FUNCTION_BLOCK ABSTRACT FB_DS402Drive IMPLEMENTS I_DS402PiezoDrive
VAR_INPUT

END_VAR
VAR_OUTPUT

END_VAR
VAR
	{attribute 'no_copy'}
    stPiezoStage		:	REFERENCE TO ST_PiezoStage;
	eDriveState			:	E_DS402DriveState;
	fbLogError			:   FB_LogMotionError;
    eHomingState		: 	E_DS402Homing;
	// reuse to absolute/relative moves for DS402
    eAxisState			:  MC_AxisStates;
    // create a property for some of these
    bExecMove			: BOOL;
    bExecHome			: BOOL;
    bPosGoal			: BOOL;
    bNegGoal			: BOOL;
    bNewMoveReq			: BOOL;
    bHomingBusy			: BOOL;
    bHomingDone			: BOOL;
    bPrepareDisable		: BOOL;
    bMoveDone			: BOOL;
    bMoveBusy			: BOOL;
	bHalted				: BOOL;
	bAborted			: BOOL;
	bStopped			: BOOL;
	bServoOffTrans	: BOOL;
	bServoOnTrans : BOOL;
	bServoOffMode		:	BOOL ;
	bServoOnMode		: BOOL;
	bDiscreteInit		: BOOL;
	bDiscreteMotionAct  : BOOL;
	bServoOffparamsSet  : BOOL;
	bServoOffparamsSetDone : BOOL;
	bLimOverride				: BOOL;

    bError				: BOOL:=FALSE;
	bErrorStop			: BOOL;
    // use this for motion time axis states
    bExecute			: BOOL;
	// This prevent unexpected logical 1 on stMotionStage.bExecute 
    nErrorId			: UDINT:=0;
    sLocalErrorMessage	: STRING;
	nPiezoErrorCode		: UDINT;
	// Save abd restore encoder value
    bInit				: BOOL;
    bLoad				: BOOL;
    bEncError			: BOOL;
	bSaveDone			: BOOL;
	bAbortDone			: BOOL;
    // axis status -- emulating some NC axis
    bClosedLoopMode		:	BOOL;
    bPositiveDirection	:  	BOOL;
    bNegativeDirection 	:  	BOOL;
    bInTargetPosition 	:  	BOOL;
	bReadErrDone			: 	BOOL;
	bLogReady			: 	BOOL;
	bFault				: 	BOOL;
    bDiscreteMotion 	:  	BOOL;
    bContinuousMotion 	:  	BOOL;

    bSlowParamReadTimer	: 	BOOL := TRUE;
	
    // Drive calibrated motion params
    nCalibratedVelocity			: DINT;
    nCalibratedAcceleration		: DINT;
    nCalibratedTargetPosition 	: DINT;
    nCalibratedMaxVelocity 		: DINT;
    nCalibratedMaxAcceleration	: DINT;
    nCalibratedHomeVelocity 	: DINT;
    nCalibratedHomeAcceleration	: DINT;

	// Open Loop Motion paramters
    nCalibratedSteps			: DINT;
    nCalibratedStepAmp			: UINT;
    nCalibratedStepFreq 		: UINT;

    // Calibrated motion params : nanometer operation by default.
    fCalibratedStandStillPos	: REAL;
    fOverride					: REAL;
	fDefaultScalingFactor 		: REAL:=0.000001;
    fCalibratedActPos			: REAL;
	rtHaltedDone	: R_TRIG;
	rtTargetReached	: R_TRIG;
	ftAbortDone: F_TRIG;
	rtFault			: R_TRIG;
    rtHomed			: R_TRIG;
    rtMoveCmdShortcut	: R_TRIG;
    rtHomeCmdShortcut	: R_TRIG;
    rtEnableMode		: R_TRIG;
    rtUserExec			: R_TRIG;
	rtErrorStop			: R_TRIG;
    rtTarget		: R_TRIG;
	rtServoOnMode	: R_TRIG;
    rtEnableDrive	: R_TRIG;
	rtServoOnTrans	: R_TRIG;
	rtNotClState 	: R_TRIG;
	rtNotOlState 	: R_TRIG;
	rtNewMoveReq	: R_TRIG;

	ftServoOffTrans	: F_TRIG;
	rtServoOffMode	: R_TRIG;
	ftAmsNetId 		: F_TRIG;
    ftExec			: F_TRIG;
	ftErrorSdoRead	: F_TRIG;
    ftEnableDrive	: F_TRIG;
	ftForwardEnabled	: F_TRIG;
	ftBackwardEnabled	: F_TRIG;
	ftServo				: F_TRIG;
	
    ftSdoStep		: 	F_TRIG;
    ftSdoStepFreq	: 	F_TRIG;
    ftSdoStepAmp	: 	F_TRIG;
	
    tonSyncHoming 		: TON;
	tonHoldTime			: TON;
	tonServoOffSync		: TON;
    tonSlowParamReadTimer: TON;
	// fast changing paramter timer -- wwe could have used PDO for this params
	// but the Piezo ESC have fixed PDO list.
	tonFastParamReadTimer: TON;
	//bInitiated	: BOOL;
    // Diagnotics data from the drive, mainly Error codes
	tRefreshDelay   : TIME := T#1S;
	tSavedholtime	: TIME;
	// Open Loop Operations
    fbSdoStep		: 	FB_EcCoESdoWrite;
    fbSdoStepFreq	: 	FB_EcCoESdoWrite;
    fbSdoStepAmp	: 	FB_EcCoESdoWrite;
	
    fbErrorSdoRead			: FB_EcCoESdoRead;
    fbFollowWinSdoRead		: FB_EcCoESdoRead;
    fbSoftLimMaxSdoRead		: FB_EcCoESdoRead;
    fbSoftLimMinSdoRead 	: FB_EcCoESdoRead;
    fbMotorloadSdoRead		: FB_EcCoESdoRead;
    fbGetAmsNetId			: FB_GetLocalAmsNetId;

    sAmsNetId 				: T_AmsNetId;
    nSubIndex  				: BYTE := 0;

  	nChanFErrWinIdx		: WORD;
  	nChanSoftwareLimIdx	: WORD;
  	nChanMotorLoadIdx	: WORD;
	nChanErrorCodeIdx	: WORD;
    nChanOlStepIdx		: WORD;
    nChanOlStepFreqIdx	: WORD;
    nChanOlStepAmpIdx	: WORD;

    nChanPrevStep			: DINT;
    nChanPrevStepFreq		: UINT;
    nChanPrevStepAmp		: UINT;

	
END_VAR


VAR CONSTANT
    nScaleOffsetBase	: WORD := 16#2007;
    nScaleInvBase		: WORD := 16#2008;
	nMotorLoadbase		: WORD := 16#200d;
    nSoftLimBase		: WORD := 16#200e;
	nHomeOffsetBase		: WORD := 16#607C;
	nHomingSpeedBase	: WORD := 16#6099;
	nhomingAccBase		: WORD := 16#609a;
	nErrorCodeBase		: WORD := 16#603f;
	nFErrWinBase		: WORD := 16#6065;
	nOlStepBase		: WORD := 16#2022;
	nOlStepAmpBase		: WORD := 16#2023;
	nOlStepFreqBase	: WORD := 16#2024;
	// this true for SmartAct MCS2 and E-727.
	nChanOfsBase	: WORD := 16#800;
	// DS 402 Motor encoder defective code : this is needed for save and restore.
	nEncErrorCode	: WORD := 16#7300;

END_VAR


VAR PERSISTENT
    bSaved: BOOL;
    fPosition: LREAL;
END_VAR

{attribute 'monitoring':= 'variable'}
PROPERTY AbortDone : BOOL
GET
AbortDone:=bAbortDone;
END_GET
SET
bAbortDone := AbortDone;
END_SET
END_PROPERTY

{attribute 'monitoring':= 'variable'}
PROPERTY Aborted : BOOL
GET
Aborted := bAborted;
END_GET
SET
bAborted := Aborted;
END_SET
END_PROPERTY

METHOD AmsNetIdToString
VAR_INPUT

END_VAR

VAR
	nCounter: UINT;
	sAmsNetTmp: STRING(255);
END_VAR
IF sAmsNetId = '' THEN
	FOR nCounter := 0 TO (SIZEOF(stPiezoStage.arNetId)-1) BY 1 DO
		IF nCounter <= ((SIZEOF(stPiezoStage.arNetId)-1) -1) THEN
			sAmsNetTmp := CONCAT(BYTE_TO_STRING(stPiezoStage.arNetId[nCounter]),'.');
		ELSE
			sAmsNetTmp := BYTE_TO_STRING(stPiezoStage.arNetId[nCounter]);
		END_IF
		sAmsNetId := CONCAT(sAmsNetId, sAmsNetTmp);
	END_FOR	
END_IF
END_METHOD

METHOD PUBLIC ABSTRACT Brake
END_METHOD

PROPERTY CalibratedAcceleration : DINT
GET
CalibratedAcceleration:=nCalibratedAcceleration;
END_GET
END_PROPERTY

PROPERTY CalibratedActPos : REAL
GET
CalibratedActPos:=fCalibratedActPos;
END_GET
END_PROPERTY

PROPERTY CalibratedHomeAcceleration : DINT
GET
CalibratedHomeAcceleration:= nCalibratedHomeVelocity;
END_GET
END_PROPERTY

PROPERTY CalibratedHomeVelocity : DINT
GET
CalibratedHomeVelocity:=nCalibratedHomeVelocity;
END_GET
END_PROPERTY

PROPERTY CalibratedMaxAcceleration : DINT
GET
CalibratedMaxAcceleration:= nCalibratedMaxAcceleration;
END_GET
END_PROPERTY

PROPERTY CalibratedMaxVelocity : DINT
GET
CalibratedMaxVelocity:= nCalibratedMaxVelocity;
END_GET
END_PROPERTY

METHOD CalibratedServoOnParams
VAR_INPUT
END_VAR
VAR

END_VAR
// All drive paramters must be express in mm, mm/s, mm/s2
nCalibratedMaxVelocity:=REAL_TO_DINT((stPiezoStage.fMaxVelocity / MAX(stPiezoStage.fscalingFactor, fDefaultScalingFactor)));
nCalibratedMaxAcceleration:=LREAL_TO_DINT(stPiezoStage.fMaxAcceleration /  MAX(stPiezoStage.fscalingFactor, fDefaultScalingFactor));
// Homing params
nCalibratedHomeVelocity:=LIMIT(0, LREAL_TO_DINT (stPiezoStage.fVelocity / MAX(stPiezoStage.fscalingFactor, fDefaultScalingFactor)), nCalibratedMaxVelocity);
nCalibratedHomeAcceleration:=LIMIT(0, LREAL_TO_DINT (stPiezoStage.fAcceleration / MAX(stPiezoStage.fscalingFactor, fDefaultScalingFactor)), nCalibratedMaxAcceleration) ;
// Target Position
nCalibratedTargetPosition:=LREAL_TO_DINT (stPiezoStage.fPosition / MAX(stPiezoStage.fscalingFactor, fDefaultScalingFactor));
// set soft limit on drive params to avoid bumping hard on the end stops
nCalibratedVelocity:=LIMIT(0, LREAL_TO_DINT (stPiezoStage.fVelocity / MAX(stPiezoStage.fscalingFactor, fDefaultScalingFactor)), nCalibratedMaxVelocity);
nCalibratedAcceleration:=LIMIT(0, LREAL_TO_DINT (stPiezoStage.fAcceleration / MAX(stPiezoStage.fscalingFactor, fDefaultScalingFactor)), nCalibratedMaxAcceleration) ;
END_METHOD

PROPERTY CalibratedTargetPosition : DINT
GET
CalibratedTargetPosition:= nCalibratedTargetPosition;
END_GET
END_PROPERTY

PROPERTY CalibratedVelocity : DINT
GET
CalibratedVelocity:=nCalibratedVelocity;
END_GET
END_PROPERTY

METHOD CalibrateServoOffParams
VAR_INPUT
END_VAR
// Open Loop Step Mode parameters
nCalibratedSteps:=LIMIT(-100000, stPiezoStage.nChanStep, 100000);
nCalibratedStepAmp:=REAL_TO_UINT(LIMIT(1, stPiezoStage.nChanStepAmp, 100) * 655.35);
nCalibratedStepFreq:=REAL_TO_UINT(LIMIT(1.0, stPiezoStage.nChanStepFreq, 1000.0));
END_METHOD

METHOD EncSaveRestore
VAR_INPUT
	bEnable	: BOOL;
END_VAR
IF bEnable THEN
    // Trigger a load if anything was saved at all
    IF NOT bInit THEN
        bInit := TRUE;
        bLoad S= bSaved;
    END_IF

    // Set our position if bLoad is true
	IF bLoad THEN
		stPiezoStage.fPosition:=fPosition;
		bSaveDone := TRUE;
	END_IF

    // Only load once, at startup
    bLoad R= bSaveDone;

    // Check ST_PiezoStage for an encoder error
    bEncError := stPiezoStage.bError AND (stPiezoStage.nErrorId = nEncErrorCode);

    // Do not save if we're currently loading or if there is an encoder error
    IF NOT bLoad AND NOT bEncError THEN
        fPosition := stPiezoStage.stAxisStatus.fActPosition;
        // This persistent variable lets us check if anything was saved
        // It will be TRUE at startup if we have saved values
        bSaved := TRUE;
    END_IF
END_IF
END_METHOD

METHOD EncValue
VAR_INPUT
  //  bEnable: BOOL;
END_VAR
(* SmartACT: The encoder count from the Piezo drive is not a raw count from the embeded actuator device
   we get a calibrated nm value. thus the use of abs() since this value is signed. 
   PI: to be discovered *)
IF stPiezoStage.nRawEncoderDINT <> 0 THEN
    stPiezoStage.nEncoderCount:=DINT_TO_UDINT(ABS(stPiezoStage.nRawEncoderDINT));
ELSE
    stPiezoStage.nEncoderCount:=0;
END_IF

// calibrated encoder readback
fCalibratedActPos:=DINT_TO_REAL(stPiezoStage.nRawEncoderDINT) *  MAX(stPiezoStage.fscalingFactor, fDefaultScalingFactor);
stPiezoStage.fPosDiff:=ABS(stPiezoStage.fPosition) - ABS(fCalibratedActPos);
END_METHOD

{attribute 'monitoring':= 'variable'}
PROPERTY Error : BOOL
GET
Error:=bError;
END_GET
SET
bError:=Error;
END_SET
END_PROPERTY

{attribute 'monitoring':= 'variable'}
PROPERTY ErrorCode : UDINT
GET
ErrorCode:=nErrorID;
END_GET
SET
nErrorID:=ErrorCode;
END_SET
END_PROPERTY

PROPERTY ErrorMessage : STRING
GET
ErrorMessage:=sLocalErrorMessage;
END_GET
SET
sLocalErrorMessage:=ErrorMessage;
END_SET
END_PROPERTY

//FB_Init is always available implicitly and it is used primarily for initialization.
//The return value is not evaluated. For a specific influence, you can also declare the
//methods explicitly and provide additional code there with the standard initialization
//code. You can evaluate the return value.
METHOD FB_Init: BOOL
VAR_INPUT
    bInitRetains: BOOL; // TRUE: the retain variables are initialized (reset warm / reset cold)
    bInCopyCode: BOOL;  // TRUE: the instance will be copied to the copy code afterward (online change)   
    stPzStage		:	REFERENCE TO ST_PiezoStage;
END_VAR
stPiezoStage REF= stPzStage;
END_METHOD

METHOD GetAmsNetId : BOOL
VAR_INPUT
	isNotSet : BOOL;
END_VAR

VAR
	
END_VAR
ftAmsNetId(CLK:=fbGetAmsNetId.bBusy);

fbGetAmsNetId(bExecute := isNotSet, tTimeOut := T#2S);

IF ftAmsNetId.Q  THEN
	IF NOT fbGetAmsNetId.bError THEN
		sAmsNetId := fbGetAmsNetId.AddrString;
	ELSE
		Error := fbGetAmsNetId.bError;
		ErrorCode := fbGetAmsNetId.nErrId;
	END_IF
	fbGetAmsNetId.bExecute := FALSE;
END_IF
END_METHOD

METHOD Halt : BOOL


Stopped S= NOT Error AND MoveBusy AND (stPiezoStage.bHalt OR NOT stPiezoStage.bExecute);

stPiezoStage.nPiezoDriveControl.8 := Stopped;
END_METHOD

{attribute 'monitoring':= 'variable'}
PROPERTY Halted : BOOL
GET
Halted := bHalted;
END_GET
SET
bHalted := Halted;
END_SET
END_PROPERTY

METHOD ABSTRACT HandleMoveRequest
VAR_INPUT
END_VAR
END_METHOD

METHOD PUBLIC Home : BOOL
tonSyncHoming(PT:=T#1000MS);
(* IMPORTANT: Homing options and parameters must be configured either via the COE online tab or via the service tool *)
CASE eHomingState OF
    E_DS402Homing.INIT_HOMING :;
        stPiezoStage.nModeOfOperation:=E_DS402OpMode.HOMING;
        IF stPiezoStage.nModeOfOperationDisplay = E_DS402OpMode.HOMING THEN
			HomeDone := FALSE;
			tonSyncHoming.IN := TRUE;
            stPiezoStage.nPiezoDriveControl.4:=TRUE;
			IF tonSyncHoming.Q THEN
				eHomingState:=E_DS402Homing.HOMING_IN_PROGRESS;
			END_IF
        END_IF

    E_DS402Homing.HOMING_IN_PROGRESS:
        IF NOT stPiezoStage.stPiezoDriveStatus.TargetReached
           AND NOT stPiezoStage.stPiezoDriveStatus.Bit13_OpModeSpecific THEN
                HomingBusy:=TRUE;
                HomeDone:=FALSE;
        END_IF
		
        // Interrupted
        IF stPiezoStage.stPiezoDriveStatus.TargetReached 
			AND NOT stPiezoStage.stPiezoDriveStatus.Bit12_OpModeSpecific THEN
            eHomingState:=E_DS402Homing.HOMING_INTERRUPTED;
        END_IF

        // Reached
        IF stPiezoStage.stPiezoDriveStatus.TargetReached
            AND stPiezoStage.stPiezoDriveStatus.Bit12_OpModeSpecific
            AND NOT stPiezoStage.stPiezoDriveStatus.Bit13_OpModeSpecific THEN
            eHomingState:=E_DS402Homing.HOMING_ATTAINED;
        END_IF

    E_DS402Homing.HOMING_ATTAINED:;
        HomingBusy:=FALSE;
        HomeDone:=TRUE;
        Error:=FALSE;
		tonSyncHoming.IN := FALSE;
		stPiezoStage.fPosition := 0.0;
		//prepare next move
		stPiezoStage.nPiezoDriveControl.4:=FALSE;
		stPiezoStage.nModeOfOperation:=E_DS402OpMode.PROFILE_POSITION;
		
    E_DS402Homing.HOMING_INTERRUPTED :;
        HomingBusy:=FALSE;
        HomeDone:=FALSE;
        ErrorMessage:='Warning: Halt interrupted homing sequence';
        Error:=FALSE;
        ErrorCode:=99; 

END_CASE
END_METHOD

{attribute 'monitoring':= 'variable'}
PROPERTY HomeDone : BOOL
GET
HomeDone:=bHomingDone;
END_GET
SET
bHomingDone:=HomeDone;
END_SET
END_PROPERTY

{attribute 'monitoring':= 'variable'}
PROPERTY HomingBusy : BOOL
GET
HomingBusy:=bHomingBusy;
END_GET
SET
bHomingBusy:=HomingBusy;
END_SET
END_PROPERTY

{attribute 'monitoring':= 'variable'}
PROPERTY PROTECTED InTargetPosition : BOOL
GET
 InTargetPosition := bInTargetPosition;
END_GET
SET
 bInTargetPosition := InTargetPosition;
END_SET
END_PROPERTY

METHOD PUBLIC Interlock

VAR
END_VAR
// Check for the plc shortcut commands
// Used for testing or to circumvent motor record issues
rtMoveCmdShortcut(CLK:=stPiezoStage.bMoveCmd);
rtHomeCmdShortcut(CLK:=stPiezoStage.bHomeCmd);

// Execute on rising edge
IF rtMoveCmdShortcut.Q AND NOT stPiezoStage.bExecute THEN
    stPiezoStage.bExecute:=TRUE;
    stPiezoStage.nCommand:=E_EpicsMotorCmd.MOVE_ABSOLUTE;
    // attempting to move an axis without homing first?
    IF stPiezoStage.nHomingMode <> E_EpicsHomeCmd.NONE AND NOT stPiezoStage.bHomed THEN
        // one can just set bHome here even though no homing was done?
        stPiezoStage.sErrorMessage:='Axis homing mode set, but homing routine pending';
    END_IF

ELSIF rtHomeCmdShortcut.Q AND NOT stPiezoStage.bExecute THEN
    stPiezoStage.bExecute:= NOT ( stPiezoStage.nCmdData = E_EpicsHomeCmd.ABSOLUTE_SET ) OR NOT ( stPiezoStage.nCmdData = E_EpicsHomeCmd.NONE);

    stPiezoStage.nCommand:=E_EpicsMotorCmd.HOME;
	// Automatically fill the correct nCmdData for homing
	stPiezoStage.nCmdData:=stPiezoStage.nHomingMode;
END_IF

// Handle main execs .  Rising on bMoved should be the ntry point
// bu this is not the case in production its a rising on bExecute.
rtUserExec(CLK:=stPiezoStage.bExecute);
// if a Move/Home Goal is comfirmed and there is no persistant 
// error conditions, then we have a valid move request.
bNewMoveReq S= NOT stPiezoStage.stAxisStatus.bBusy AND rtUserExec.Q AND NOT stPiezoStage.bError;
// this Move request is valid till an error occurs or the currently move is done
bNewMoveReq R= NOT stPiezoStage.bExecute OR stPiezoStage.bError;
bPrepareDisable R= bNewMoveReq;
// define this R_TRIG to comfirm a new move request.
rtNewMoveReq(CLK:=bNewMoveReq);
// Moves are automatically allowed if no safety hooks. Otherwise, some other code will set this.
stPiezoStage.bSafetyReady S= stPiezoStage.bPowerSelf;

// Transition to DURING_MOTION drive mode
rtEnableMode(CLK:=(stPiezoStage.nEnableMode = E_StageEnableMode.DURING_MOTION));
// Handle auto-enable timing
CASE stPiezoStage.nEnableMode OF
    E_StageEnableMode.ALWAYS:
        stPiezoStage.bEnable:=TRUE;
    E_StageEnableMode.DURING_MOTION:
		IF rtEnableMode.Q THEN
			stPiezoStage.bEnable := FALSE;
		END_IF
		// Power only enabled with a new move request
		IF rtNewMoveReq.Q THEN
			stPiezoStage.bEnable S= stPiezoStage.bSafetyReady;
		END_IF
END_CASE

bPosGoal  S= rtNewMoveReq.Q AND (stPiezoStage.stAxisStatus.fActPosition < stPiezoStage.fPosition) ;
bNegGoal  S= rtNewMoveReq.Q AND (stPiezoStage.stAxisStatus.fActPosition > stPiezoStage.fPosition) ;

bPosGoal  R= HomingBusy OR bNegGoal;
bNegGoal  R= HomingBusy OR bPosGoal;
// use falling trigger to avoid spaming  sErrorMessage
ftForwardEnabled(CLK:=stPiezoStage.bAllForwardEnable);
ftBackwardEnabled(CLK:=stPiezoStage.bAllBackwardEnable);

IF  NOT HomingBusy AND ftForwardEnabled.Q THEN
	// Not an error, just a warning
	stPiezoStage.sErrorMessage:='Cannot move past positive limit.';
	bLimOverride := TRUE;
	stPiezoStage.bExecute:=FALSE;
END_IF
	
IF NOT HomingBusy AND ftBackwardEnabled.Q THEN
	// Not an error, just a warning
	stPiezoStage.sErrorMessage:='Cannot move past Negative limit.';
	bLimOverride := TRUE;
	stPiezoStage.bExecute:=FALSE;
END_IF

IF NOT stPiezoStage.bError AND stPiezoStage.bExecute AND NOT stPiezoStage.bUserEnable THEN
    stPiezoStage.bError := TRUE;
    stPiezoStage.nErrorId := 1;
    stPiezoStage.sCustomErrorMessage := 'Move requested, but user enable is disabled!';
END_IF

// Update all enable booleans
SetEnables();

CASE McAxisState OF
    // We are not enabled if there is an issue
    MC_AXISSTATE_UNDEFINED, MC_AXISSTATE_DISABLED, MC_AXISSTATE_ERRORSTOP:
        stPiezoStage.bEnableDone:=FALSE;
    ELSE
        stPiezoStage.bEnableDone:=TRUE;
END_CASE

bExecute:= NOT stPiezoStage.bError AND stPiezoStage.bExecute AND stPiezoStage.bAllEnable AND stPiezoStage.bEnableDone AND stPiezoStage.bSafetyReady;
// 
bExecHome:=bExecute AND stPiezoStage.nCommand = 10;
bExecMove:=bExecute AND NOT bExecHome;

(*  *)
ftExec(CLK:=stPiezoStage.bExecute);
END_METHOD

METHOD PUBLIC Logger
END_METHOD

{attribute 'monitoring':= 'variable'}
PROPERTY McAxisState : MC_AxisStates
GET
McAxisState := eAxisState;
END_GET
SET
eAxisState := McAxisState;
END_SET
END_PROPERTY

METHOD PUBLIC  MotionParams
VAR_INPUT
    tRefreshDelay: TIME;
END_VAR
// get periodique update on Motion params
ReadDriveParams();
// 
// Copy axis parameters that we want to expose to the EPICS layer.
stPiezoStage.stAxisParametersExposed.bCtrlEnablePosDiffControl     := stPiezoStage.stAxisParameters.bCtrlEnablePosDiffControl;
stPiezoStage.stAxisParametersExposed.bEncEnableSoftEndMaxControl   := stPiezoStage.stAxisParameters.bEncEnableSoftEndMaxControl ;
stPiezoStage.stAxisParametersExposed.bEncEnableSoftEndMinControl   := stPiezoStage.stAxisParameters.bEncEnableSoftEndMinControl;
stPiezoStage.stAxisParametersExposed.fAccelerationMax              := stPiezoStage.stAxisParameters.fAccelerationMax;
stPiezoStage.stAxisParametersExposed.fCtrlPosDiffMax               := stPiezoStage.stAxisParameters.fCtrlPosDiffMax;
stPiezoStage.stAxisParametersExposed.fCtrlPosDiffMaxTime           := stPiezoStage.stAxisParameters.fCtrlPosDiffMaxTime;
stPiezoStage.stAxisParametersExposed.fDecelerationMax              := stPiezoStage.stAxisParameters.fDecelerationMax;
stPiezoStage.stAxisParametersExposed.fEncSoftEndMax                := stPiezoStage.stAxisParameters.fEncSoftEndMax;
stPiezoStage.stAxisParametersExposed.fEncSoftEndMin                := stPiezoStage.stAxisParameters.fEncSoftEndMin;
stPiezoStage.stAxisParametersExposed.fVeloMaximum                  := stPiezoStage.stAxisParameters.fVeloMaximum;
stPiezoStage.stAxisParametersExposed.fEncOffset               	  := stPiezoStage.stAxisParameters.fEncOffset;
stPiezoStage.stAxisParametersExposed.fEncScaleFactorInternal       := stPiezoStage.stAxisParameters.fEncScaleFactorInternal;
END_METHOD

METHOD PUBLIC ABSTRACT MoveAbsolute
END_METHOD

{attribute 'monitoring':= 'variable'}
PROPERTY MoveBusy : BOOL
GET
MoveBusy:=bMoveBusy;
END_GET
SET
bMoveBusy:=MoveBusy;
END_SET
END_PROPERTY

{attribute 'monitoring':= 'variable'}
PROPERTY MoveDone : BOOL
GET
MoveDone:=bMoveDone;
END_GET
SET
bMoveDone:=MoveDone;
END_SET
END_PROPERTY

METHOD PUBLIC ABSTRACT MoveRelative
VAR_INPUT
END_VAR
END_METHOD

METHOD PUBLIC ABSTRACT MoveVelocity
END_METHOD

{attribute 'monitoring':= 'variable'}
PROPERTY PiezoErrorCode : UDINT
GET
PiezoErrorCode := nPiezoErrorCode;
END_GET
SET
nPiezoErrorCode := PiezoErrorCode;
END_SET
END_PROPERTY

METHOD PostInterlocks
VAR_INPUT
END_VAR
// user override aka stop from EPICS ?
// Check done moving via user stop, fbDriveVirtual and Target Position Monitoring, or from homing.
// set/reset stPiezoStage.bDone after move absolute/Relative

// need to catch this as soon as it happen and must be seen by every call after intelock()
// within the sma ecycle
ftAbortDone(CLK:=AbortDone);
//rtErrorStop(CLK:=bErrorStop);

rtTarget(CLK:=(InTargetPosition AND MoveDone AND bExecMove));
rtHomed(CLK:=HomeDone AND bExecHome);
IF (*rtErrorStop.Q OR*) ftAbortDone.Q OR  rtTarget.Q OR rtHomed.Q THEN
    IF NOT stPiezoStage.bDone THEN
		MoveBusy:=FALSE;
		stPiezoStage.bDone := MoveDone OR HomeDone;
		stPiezoStage.bHomed := HomeDone;
		AbortDone := FALSE;
		bErrorStop:=FALSE;
        IF NOT Error THEN
            bExecute:=FALSE;
            stPiezoStage.bExecute:=FALSE;
        END_IF
    END_IF
END_IF

IF bExecute AND NOT Error THEN
    // Reset local warnings if things are going well
    stPiezoStage.sErrorMessage:='';
END_IF

// Handle auto-disable timing
bPrepareDisable S= stPiezoStage.nEnableMode = E_StageEnableMode.DURING_MOTION AND ftExec.Q;
// Delay the disable until we reach standstill, else brake issues or other race conditions
IF bPrepareDisable AND eAxisState = MC_AXISSTATE_STANDSTILL THEN
    bPrepareDisable:=FALSE;
    stPiezoStage.bEnable:=FALSE;
END_IF

//---------- brakes code here ---------------

// Always reset, even if not rising edge, so command can be issued again
// but do so only after the move was done or was cancel due to error or an interlock condition
IF ftExec.Q AND (stPiezoStage.bMoveCmd OR stPiezoStage.bHomeCmd) THEN
    stPiezoStage.bMoveCmd:=FALSE;
    stPiezoStage.bHomeCmd:=FALSE;

END_IF

// Force everything off in case of error
IF stPiezoStage.bError THEN
    stPiezoStage.bBusy := FALSE;
    stPiezoStage.bDone := FALSE;
    stPiezoStage.bEnable := FALSE;
END_IF

stPiezoStage.bBusy:=HomingBusy OR MoveBusy;

// Log errors
// Set the error message if we have one

// Hook if other code wants to inject a non-NC error
IF stPiezoStage.sCustomErrorMessage <> '' THEN
	bLogReady := FALSE;
	stPiezoStage.sErrorMessage := stPiezoStage.sCustomErrorMessage;

ELSE
	stPiezoStage.sErrorMessage := F_MotionErrorCodeLookup(nErrorId := stPiezoStage.nErrorId);
END_IF

fbLogError( stMotionStage:=stPiezoStage, bEnable:=bLogReady);
END_METHOD

METHOD Power : BOOL
// No transition while the drive is in motion
// transition from close to open loop. while moving

rtEnableDrive(CLK:=stPiezoStage.bAllEnable);
ftEnableDrive(CLK:=stPiezoStage.bAllEnable);

ftServoOffTrans(CLK:=(NOT bFault AND stPiezoStage.bServo));
rtServoOnTrans(CLK:=(NOT bFault AND stPiezoStage.bServo));

//rtServoOffMode(CLK:=bServoOffMode);
//rtServoOnMode(CLK:=stPiezoStage.bAllEnable AND bServoOnMode);
// Enabled the drive: the client code must wait for state transition.
IF (bServoOffMode OR bServoOnMode) AND rtEnableDrive.Q THEN
    // Voltage on, close loop operations
    stPiezoStage.nPiezoDriveControl:=16#0F;
    fOverride:=100.0;
	
ELSIF ftEnableDrive.Q (*OR rtServoOffMode.Q*) THEN
	//  inhibit motion functions! keep amplifier enable
	stPiezoStage.nPiezoDriveControl:=16#07;
    fOverride:=0.0;
ELSE
	;
END_IF

IF bServoOffTrans AND ( stPiezoStage.nModeOfOperationDisplay = E_DS402OpMode.MCS2_OL_SM ) THEN
	// ready for open loop operation
	bServoOffTrans := FALSE;
	bServoOffMode := TRUE;
	bServoOnMode := FALSE;
ELSIF bServoOnTrans AND ( stPiezoStage.nModeOfOperationDisplay = E_DS402OpMode.PROFILE_POSITION ) THEN
	// ready for closed loop operation
	bServoOnTrans := FALSE;
	bServoOffMode := FALSE;
	bServoOnMode := TRUE;
	
ELSIF ftServoOffTrans.Q THEN
	bServoOffTrans := TRUE;
	bServoOnTrans := FALSE;
	stPiezoStage.nModeOfOperation := E_DS402OpMode.MCS2_OL_SM;
	
// transition to close loop mode
ELSIF rtServoOnTrans.Q THEN
	bServoOffTrans := FALSE;
	bServoOnTrans := TRUE;
	stPiezoStage.nModeOfOperation := E_DS402OpMode.PROFILE_POSITION;
END_IF



// rtNotClState(CLK:=(eDriveState <> E_DS402DriveState.OPERATION_ENABLED));
// rtNotOlState(CLK:=(eDriveState <> E_DS402DriveState.SWITCH_ON));
// 
// IF rtNotClState.Q THEN
// 	bClosedLoopMode := FALSE;
// ELSIF rtNotOlState.Q THEN 
// 	bOpenLoopMode := FALSE;
// ELSIF rtNotClState.Q AND rtNotOlState.Q THEN
// 	McAxisState:=MC_AxisStates.MC_AXISSTATE_DISABLED;
// END_IF
END_METHOD

METHOD ReadDriveErrors : BOOL
VAR_INPUT

END_VAR

VAR

END_VAR
//AmsNetIdToString();

ftErrorSdoRead(CLK:=fbErrorSdoRead.bBusy);

fbErrorSdoRead( sNetId:= sAmsNetId, 
				nSlaveAddr:=stPiezoStage.nSlaveAddr, 
				nIndex:=nChanErrorCodeIdx, 
				nSubIndex :=nSubIndex, 
				pDstBuf:= ADR(nPiezoErrorCode), 
				cbBufLen:=SIZEOF(nPiezoErrorCode),
				bExecute:= Error );
				
IF ftErrorSdoRead.Q THEN
	IF 	fbErrorSdoRead.bError THEN
		Error:=fbErrorSdoRead.bError;
		ErrorCode:=fbErrorSdoRead.nErrId;
	ELSE
		// Update Motion Error code;
		ErrorCode := PiezoErrorCode;
		stPiezoStage.bError := Error;
		stPiezoStage.nErrorId := ErrorCode;	
		bLogReady := TRUE;
	END_IF
	ReadDriveErrors := TRUE;
ELSE
	ReadDriveErrors := FALSE;
END_IF

//ReadDriveErrors := bReadErrDone;
END_METHOD

(*Read Piezo drive Motion parameters*)
METHOD ReadDriveParams : BOOL
VAR_INPUT

END_VAR

VAR
END_VAR
tonSlowParamReadTimer( IN:=bSlowParamReadTimer, PT:=tRefreshDelay );
AmsNetIdToString();

// Get the following Error
fbFollowWinSdoRead(	sNetId:= sAmsNetId, 
				nSlaveAddr:=stPiezoStage.nSlaveAddr, 
				nIndex:=nChanFErrWinIdx, 
				nSubIndex:=0, 
				pDstBuf:= ADR(stPiezoStage.nfErrWin), 
				cbBufLen:=SIZEOF(stPiezoStage.nfErrWin),
				bExecute:=tonSlowParamReadTimer.Q
			  );
// Read the Upper software limit
fbSoftLimMaxSdoRead( sNetId:= sAmsNetId, 
				nSlaveAddr:=stPiezoStage.nSlaveAddr, 
				nIndex:=nChanSoftwareLimIdx, 
				nSubIndex:=1, 
				pDstBuf:= ADR(stPiezoStage.nSoftLimMax), 
				cbBufLen:=SIZEOF(stPiezoStage.nSoftLimMax),
				bExecute:=tonSlowParamReadTimer.Q
			  );
		  
// Read the Lower software limit		  
fbSoftLimMinSdoRead( sNetId:= sAmsNetId, 
				nSlaveAddr:=stPiezoStage.nSlaveAddr, 
				nIndex:=nChanSoftwareLimIdx, 
				nSubIndex:=2, 
				pDstBuf:= ADR(stPiezoStage.nSoftLimMin), 
				cbBufLen:=SIZEOF(stPiezoStage.nSoftLimMin),
				bExecute:=tonSlowParamReadTimer.Q
			  );

IF fbSoftLimMinSdoRead.bBusy AND fbSoftLimMaxSdoRead.bBusy AND fbFollowWinSdoRead.bBusy THEN
	bSlowParamReadTimer:=FALSE;
END_IF

IF NOT fbSoftLimMinSdoRead.bBusy AND NOT fbSoftLimMaxSdoRead.bBusy AND NOT fbFollowWinSdoRead.bBusy THEN
	IF NOT bSlowParamReadTimer THEN
		bSlowParamReadTimer:=TRUE;
	END_IF
	IF 	fbFollowWinSdoRead.bError THEN
		// this will be logged as a warning
		Error := FALSE;
		PiezoErrorCode := fbFollowWinSdoRead.nErrId;
		//fbMotionErrorLogger.AddMsg(PiezoErrorCode, '');
	ELSIF 	fbSoftLimMaxSdoRead.bError THEN
		// this will be logged as a warning
		Error := FALSE;
		PiezoErrorCode := fbSoftLimMaxSdoRead.nErrId;
		//fbMotionErrorLogger.AddMsg(PiezoErrorCode, '');
	ELSIF 	fbSoftLimMinSdoRead.bError THEN
		// this will be logged as a warning
		Error := FALSE;
		PiezoErrorCode := fbSoftLimMinSdoRead.nErrId;
		//fbMotionErrorLogger.AddMsg(PiezoErrorCode, '');
	END_IF
	stPiezoStage.bError := Error;
	stPiezoStage.nErrorId := PiezoErrorCode;
END_IF

stPiezoStage.stAxisParameters.sAxisName := stPiezoStage.sName;
stPiezoStage.stAxisParameters.AxisId := stPiezoStage.nMotionAxisID;
stPiezoStage.stAxisParameters.bCtrlEnablePosDiffControl   := BOOL_TO_WORD(stPiezoStage.nfErrWin > 0);
stPiezoStage.stAxisParameters.bEncEnableSoftEndMaxControl := BOOL_TO_WORD(stPiezoStage.nSoftLimMax > stPiezoStage.nSoftLimMin);
stPiezoStage.stAxisParameters.bEncEnableSoftEndMinControl := BOOL_TO_WORD(stPiezoStage.nSoftLimMin < stPiezoStage.nSoftLimMax);
stPiezoStage.stAxisParameters.fAccelerationMax := stPiezoStage.fMaxAcceleration;
stPiezoStage.stAxisParameters.fCtrlPosDiffMax := stPiezoStage.nfErrWin;
// this info is not provided by the drive we keep it 0
stPiezoStage.stAxisParameters.fCtrlPosDiffMaxTime := 0.0;
stPiezoStage.stAxisParameters.fDecelerationMax := stPiezoStage.fMaxAcceleration;
stPiezoStage.stAxisParameters.fEncSoftEndMax := LINT_TO_LREAL(stPiezoStage.nSoftLimMax);
stPiezoStage.stAxisParameters.fEncSoftEndMin := LINT_TO_LREAL(stPiezoStage.nSoftLimMin);
stPiezoStage.stAxisParameters.fVeloMaximum := stPiezoStage.fMaxVelocity;
stPiezoStage.stAxisParameters.fEncOffset := 0.0;
// this info is not provided by the driver we keep it 0
stPiezoStage.stAxisParameters.fEncScaleFactorInternal := 0.0;
stPiezoStage.bAxisParamsInit S= TRUE;
END_METHOD

METHOD Reset : BOOL
// Try to clear any faults if they are present by setting bit 7 of the Control Word.
IF stPiezoStage.bReset THEN
    stPiezoStage.nPiezoDriveControl:=16#80;
    // Reset everything when bReset is flagged
    stPiezoStage.bEnable:=FALSE;
    stPiezoStage.bReset:=FALSE;
    stPiezoStage.bExecute:=FALSE;
	Error := FALSE;
	ErrorCode := 0;
	PiezoErrorCode := 0;
	stPiezoStage.bError := 0;
	stPiezoStage.nErrorId := 0;	
    stPiezoStage.sErrorMessage:='';
    stPiezoStage.sCustomErrorMessage:='';
    bExecute:=FALSE;
	bLogReady := FALSE;
	HomeDone := FALSE;
	// Need to clear this when htting endstop
	MoveBusy := FALSE;
END_IF
END_METHOD

METHOD SetEnables
VAR_INPUT
END_VAR
stPiezoStage.bAllForwardEnable:=stPiezoStage.bLimitForwardEnable AND (stPiezoStage.bGantryForwardEnable OR NOT stPiezoStage.bGantryAxis) AND stPiezoStage.stEPSForwardEnable.bEPS_OK;
stPiezoStage.bAllBackwardEnable:=stPiezoStage.bLimitBackwardEnable AND (stPiezoStage.bGantryBackwardEnable OR NOT stPiezoStage.bGantryAxis) AND stPiezoStage.stEPSBackwardEnable.bEPS_OK;

stPiezoStage.bAllEnable:=stPiezoStage.bEnable AND stPiezoStage.bHardwareEnable AND stPiezoStage.stEPSPowerEnable.bEPS_OK;
stPiezoStage.bAllEnable R= NOT stPiezoStage.bUserEnable;
END_METHOD

METHOD SetServoOffParams : BOOL
VAR_INPUT

END_VAR
IF THIS^.bServoOffMode THEN
AmsNetIdToString();

fbSdoStep(
    sNetId     := sAmsNetId,
    nSlaveAddr := stPiezoStage.nSlaveAddr,
    nIndex     := nChanOlStepIdx,
    nSubIndex  := 0,
    pSrcBuf    := ADR(nCalibratedSteps),
    cbBufLen   := SIZEOF(stPiezoStage.nChanStep),
    bExecute   := bServoOffparamsSet
);

fbSdoStepAmp(
    sNetId     := sAmsNetId,
    nSlaveAddr := stPiezoStage.nSlaveAddr,
    nIndex     := nChanOlStepAmpIdx,
    nSubIndex  := 0,
    pSrcBuf    := ADR(nCalibratedStepAmp),
    cbBufLen   := SIZEOF(stPiezoStage.nChanStepAmp),
    bExecute   := bServoOffparamsSet
);

fbSdoStepFreq(
    sNetId     := sAmsNetId,
    nSlaveAddr := stPiezoStage.nSlaveAddr,
    nIndex     := nChanOlStepFreqIdx,
    nSubIndex  := 0,
    pSrcBuf    := ADR(nCalibratedStepFreq),
    cbBufLen   := SIZEOF(stPiezoStage.nChanStepFreq),
    bExecute   := bServoOffparamsSet
);

// ftSdoStep(CLK:=fbSdoStep.bBusy);
// ftSdoStepFreq(CLK:=fbSdoStepAmp.bBusy);
// ftSdoStepAmp(CLK:=fbSdoStepFreq.bBusy);
// 
// IF ftSdoStep.Q AND ftSdoStepFreq.Q AND ftSdoStepAmp.Q THEN
IF NOT fbSdoStep.bBusy AND NOT fbSdoStepAmp.bBusy AND NOT fbSdoStepFreq.bBusy THEN
	IF 	fbSdoStep.bError THEN
		// this will be logged as a warning
		Error := FALSE;
		PiezoErrorCode := fbSdoStep.nErrId;
		//fbMotionErrorLogger.AddMsg(PiezoErrorCode, '');
	ELSIF fbSdoStepAmp.bError THEN
		// this will be logged as a warning
		Error := FALSE;
		PiezoErrorCode := fbSdoStepAmp.nErrId;
		//fbMotionErrorLogger.AddMsg(PiezoErrorCode, '');
	ELSIF fbSdoStepFreq.bError THEN
		// this will be logged as a warning
		Error := FALSE;
		PiezoErrorCode := fbSdoStepFreq.nErrId;
		//fbMotionErrorLogger.AddMsg(PiezoErrorCode, '');
	END_IF
	stPiezoStage.bError := Error;
	stPiezoStage.nErrorId := PiezoErrorCode;
	IF Error THEN
		bServoOffparamsSetDone := FALSE;
	END_IF
	bServoOffparamsSet := FALSE;
	bServoOffparamsSetDone := TRUE;
	nChanPrevStep := stPiezoStage.nChanStep;
	nChanPrevStepAmp := stPiezoStage.nChanStepAmp;
	nChanPrevStepFreq := stPiezoStage.nChanStepFreq;
END_IF

END_IF
SetServoOffParams := bServoOffparamsSetDone;
END_METHOD

METHOD StateMachine
VAR_INPUT
END_VAR
rtFault(CLK:=bFault	);

(*switch on disable*)
IF NOT stPiezoStage.stPiezoDriveStatus.ReadyToSwitchOn
    AND NOT stPiezoStage.stPiezoDriveStatus.SwitchedOn
    AND NOT stPiezoStage.stPiezoDriveStatus.OperationEnabled
    AND NOT stPiezoStage.stPiezoDriveStatus.Fault
    AND stPiezoStage.stPiezoDriveStatus.VoltageEnabled
    AND NOT stPiezoStage.stPiezoDriveStatus.QuickStopActive
    AND  stPiezoStage.stPiezoDriveStatus.SwitchOnDisabled THEN

    eDriveState :=E_DS402DriveState.SWITCH_ON_DISABLED;
END_IF

(*Ready to switch*)
IF stPiezoStage.stPiezoDriveStatus.ReadyToSwitchOn
    AND NOT stPiezoStage.stPiezoDriveStatus.SwitchedOn
    AND NOT stPiezoStage.stPiezoDriveStatus.OperationEnabled
    AND NOT stPiezoStage.stPiezoDriveStatus.Fault
    AND stPiezoStage.stPiezoDriveStatus.VoltageEnabled
    AND stPiezoStage.stPiezoDriveStatus.QuickStopActive
    AND NOT stPiezoStage.stPiezoDriveStatus.SwitchOnDisabled THEN
	
	bFault := FALSE;
    eDriveState :=E_DS402DriveState.SWITCH_ON_READY;
END_IF

(*Switch on*)
IF stPiezoStage.stPiezoDriveStatus.ReadyToSwitchOn
    AND  stPiezoStage.stPiezoDriveStatus.SwitchedOn
    AND NOT stPiezoStage.stPiezoDriveStatus.OperationEnabled
    AND NOT stPiezoStage.stPiezoDriveStatus.Fault
    AND stPiezoStage.stPiezoDriveStatus.VoltageEnabled
    AND stPiezoStage.stPiezoDriveStatus.QuickStopActive
    AND NOT stPiezoStage.stPiezoDriveStatus.SwitchOnDisabled THEN

    eDriveState :=E_DS402DriveState.SWITCH_ON;
END_IF

(*Operation enbaled*)
IF stPiezoStage.stPiezoDriveStatus.ReadyToSwitchOn
    AND stPiezoStage.stPiezoDriveStatus.SwitchedOn
    AND stPiezoStage.stPiezoDriveStatus.OperationEnabled
    AND NOT stPiezoStage.stPiezoDriveStatus.Fault
    AND stPiezoStage.stPiezoDriveStatus.VoltageEnabled
    AND stPiezoStage.stPiezoDriveStatus.QuickStopActive
    AND NOT stPiezoStage.stPiezoDriveStatus.SwitchOnDisabled THEN

    eDriveState :=E_DS402DriveState.OPERATION_ENABLED;
END_IF

(*Quick Stop: Note used for MCS2*) 
IF stPiezoStage.stPiezoDriveStatus.ReadyToSwitchOn
    AND stPiezoStage.stPiezoDriveStatus.SwitchedOn
    AND stPiezoStage.stPiezoDriveStatus.OperationEnabled
    AND NOT stPiezoStage.stPiezoDriveStatus.Fault
    AND stPiezoStage.stPiezoDriveStatus.VoltageEnabled
    AND NOT stPiezoStage.stPiezoDriveStatus.QuickStopActive
    AND NOT stPiezoStage.stPiezoDriveStatus.SwitchOnDisabled THEN

    eDriveState :=E_DS402DriveState.QUICK_STOP_ACTIVE;
END_IF

(*Fault*)
IF  NOT stPiezoStage.stPiezoDriveStatus.ReadyToSwitchOn
    AND NOT stPiezoStage.stPiezoDriveStatus.SwitchedOn
    AND NOT stPiezoStage.stPiezoDriveStatus.OperationEnabled
    AND stPiezoStage.stPiezoDriveStatus.Fault
    AND stPiezoStage.stPiezoDriveStatus.VoltageEnabled
    AND NOT stPiezoStage.stPiezoDriveStatus.QuickStopActive
    AND NOT stPiezoStage.stPiezoDriveStatus.SwitchOnDisabled THEN
	bFault := TRUE;
    eDriveState :=E_DS402DriveState.FAULT;
END_IF



CASE eDriveState  OF

    E_DS402DriveState.SWITCH_ON_DISABLED:;
		bFault := FALSE;
    E_DS402DriveState.SWITCH_ON_READY:;
		bFault := FALSE;
    E_DS402DriveState.SWITCH_ON:;
		// catch most recent motion error
		IF Error THEN
			McAxisState:=MC_AxisStates.MC_AXISSTATE_ERRORSTOP;
		END_IF
		
    E_DS402DriveState.OPERATION_ENABLED:;
		IF (bServoOffMode OR bServoOnMode) AND NOT THIS^.MoveBusy THEN
			McAxisState:=MC_AxisStates.MC_AXISSTATE_STANDSTILL;
		END_IF
		
    E_DS402DriveState.FAULT:;
        (* This is not a motion fault but rather a hardware, lost of enabled, wc or loss of calibration issue
			The condition will set bit 3 'fault' but not bit 13 'error' so waiting in the error state would won't  clear this condition *)
		IF rtFault.Q THEN
			Error := TRUE;
			McAxisState:=MC_AxisStates.MC_AXISSTATE_UNDEFINED;
		END_IF
		// Catch the drive errors code
		ReadDriveErrors();

    E_DS402DriveState.QUICK_STOP_ACTIVE:;


END_CASE
END_METHOD

{attribute 'monitoring':= 'variable'}
PROPERTY Stopped : BOOL
GET
Stopped:=bStopped;
END_GET
SET
bStopped := Stopped;
END_SET
END_PROPERTY

PROPERTY PUBLIC stPzStage : REFERENCE TO ST_PiezoStage
SET
THIS^.stPiezoStage REF= stPzStage;
END_SET
END_PROPERTY

METHOD SyncEpicsStatus
VAR_INPUT
END_VAR
//Status struct for EPICS communication
stPiezoStage.stAxisStatus.bEnable:=stPiezoStage.bAllEnable;
stPiezoStage.stAxisStatus.bEnabled:=stPiezoStage.bEnableDone; // account for PowerEnable from power block
stPiezoStage.stAxisStatus.bError:=stPiezoStage.bError;
stPiezoStage.stAxisStatus.bHomeSensor:=stPiezoStage.bHome;
stPiezoStage.stAxisStatus.bLimitBwd:=stPiezoStage.bAllBackwardEnable;
stPiezoStage.stAxisStatus.bLimitFwd:=stPiezoStage.bAllForwardEnable;
stPiezoStage.stAxisStatus.bReset:=stPiezoStage.bReset;
stPiezoStage.stAxisStatus.fAcceleration:=stPiezoStage.fAcceleration;
stPiezoStage.stAxisStatus.fActDiff:=stPiezoStage.fPosDiff;
stPiezoStage.stAxisStatus.fActPosition:=THIS^.CalibratedActPos;
stPiezoStage.stAxisStatus.fActVelocity:=stPiezoStage.fVelocity;
stPiezoStage.stAxisStatus.fDeceleration:=stPiezoStage.fAcceleration;
stPiezoStage.stAxisStatus.fOverride:=THIS^.fOverride;
stPiezoStage.stAxisStatus.fPosition:=stPiezoStage.fPosition;
stPiezoStage.stAxisStatus.fVelocity:=stPiezoStage.fVelocity;
stPiezoStage.stAxisStatus.nCmdData:=stPiezoStage.nCmdData;  //Or nCmdDataLocal
stPiezoStage.stAxisStatus.nCommand:=stPiezoStage.nCommand;  //Or nCommandLocal
stPiezoStage.stAxisStatus.nErrorId:=stPiezoStage.nErrorId;
stPiezoStage.stAxisStatus.bBusy:=stPiezoStage.bBusy;
stPiezoStage.stAxisStatus.bHomed:=stPiezoStage.bHomed;
stPiezoStage.stAxisStatus.bExecute:=bExecute;
stPiezoStage.stAxisStatus.nCommand:=3; // If this is not 3, the IOC stops updating positions during homing
END_METHOD

END_FUNCTION_BLOCK

(* stored: Version 1.1.0.1
   POU FB_DS402Drive: Id {062edea9-cfc5-43cf-98da-5ad9b4d99528}, SpecialFunc None
   Property AbortDone: Id {784ddc4a-64d1-4d90-874b-4cd96de2c7ff}
   Get Get: Id {6999c219-a1cd-49cb-894a-c97e03b5a02c}
   Set Set: Id {9ef94df7-19a3-4100-9562-779a33e78842}
   Property Aborted: Id {3fe65c2b-824e-4981-9c1c-69f25158ffa6}
   Get Get: Id {b5738d0e-f4d1-4805-85b8-287b01d2eb55}
   Set Set: Id {9d75ef58-86dd-47b9-85ee-3172ec9e9c5a}
   Method AmsNetIdToString: Id {7c03e2af-a3ad-4f9f-ae86-d47bb3a86f54}
   Method Brake: Id {c6b36a48-c7b1-4cfe-936b-d492d651f479}
   Property CalibratedAcceleration: Id {c9db77b1-cfd0-4d09-b550-344bf9246222}
   Get Get: Id {0de4f123-8d8a-4161-9634-33cbec6d4458}
   Property CalibratedActPos: Id {f59b6d0c-3ed5-49c8-8c42-f3fe81b218e0}
   Get Get: Id {7008e174-6003-4a34-8527-bc95fa10dfd5}
   Property CalibratedHomeAcceleration: Id {c1c6c121-0b12-42af-974e-2797f2c4272d}
   Get Get: Id {8d5efd04-0b17-46db-97b7-cc2c95fa3465}
   Property CalibratedHomeVelocity: Id {c44daf34-c381-47a9-8593-74a52579bfbc}
   Get Get: Id {9eff9bf5-b655-4dd6-b1a5-19a4350b2a68}
   Property CalibratedMaxAcceleration: Id {3c0a3332-3cbc-4bab-89e4-c4f12fcb17c6}
   Get Get: Id {2bce7c96-ff01-4efa-aa37-c5c3266f5a5e}
   Property CalibratedMaxVelocity: Id {6dc4e13f-94e3-4e5c-88a6-b12b64a1e91a}
   Get Get: Id {f99c53d5-5340-4fb2-aeed-beb7f587e2c8}
   Method CalibratedServoOnParams: Id {ac17b7c4-a540-4db8-be71-88c2b2fc9fb9}
   Property CalibratedTargetPosition: Id {81813abc-be79-4b01-bd0b-013ad1ba8c86}
   Get Get: Id {b29f2fdd-a221-4a00-b566-55ff2dd3354a}
   Property CalibratedVelocity: Id {54e27d08-db1c-4a56-8d6f-ee25264ddf78}
   Get Get: Id {55f6b951-9e85-4976-9d4e-affbfb1a904d}
   Method CalibrateServoOffParams: Id {c9ba05b5-4e10-4360-a86f-570163826c05}
   Method EncSaveRestore: Id {62326dfa-915c-4ff5-a6ba-aedff0abd839}
   Method EncValue: Id {f460e6f3-54f0-4341-b7f0-33fb3e421551}
   Property Error: Id {6f16c5a8-a341-41d8-bb67-663d3f8d4084}
   Get Get: Id {b7c85154-eaf9-42ce-80df-d89782c46cda}
   Set Set: Id {2447c241-763d-4843-985e-1e7b2b4157d6}
   Property ErrorCode: Id {a05ec7b2-e4fa-4c9a-9ffa-8d608185c857}
   Get Get: Id {5d902389-8aa3-41b0-82ce-2f29a350e020}
   Set Set: Id {8d492092-46f5-4d0a-b5a1-6972c25ffd11}
   Property ErrorMessage: Id {234fb137-8bc4-42b9-a4b9-3f1687c56fcc}
   Get Get: Id {875ab620-c818-4cc8-91f8-7ebc15876b2a}
   Set Set: Id {3b380431-6fb8-4f07-bb22-d7ab556e09f5}
   Method FB_Init: Id {71e69160-f135-4315-a4e8-cd410a533efe}
   Method GetAmsNetId: Id {599152ff-bf5a-4de5-82dd-edaef94bc45d}
   Method Halt: Id {7f626c89-4c25-446a-aadf-2d7158be6cb2}
   Property Halted: Id {e29ce96f-0218-49b1-9df6-38964ec70373}
   Get Get: Id {1f59584f-779f-4818-a936-530be93a244e}
   Set Set: Id {b6e4320c-ca7d-46e3-bd9d-374bb4de7cc9}
   Method HandleMoveRequest: Id {ff2773a0-e7b2-4853-a67a-3829c631e808}
   Method Home: Id {2fdfc142-a2a6-49f0-950a-d0e52b5408ca}
   Property HomeDone: Id {ef80f79d-a7a5-4a2f-a11f-e37d59b9ba61}
   Get Get: Id {742e7703-4c8b-4cae-8b7c-4c09294b165f}
   Set Set: Id {a950124f-24af-4212-9907-e7e43ac15290}
   Property HomingBusy: Id {68d84e73-fc8a-4bd0-8abf-2cf5ca63e71e}
   Get Get: Id {90949a4e-2ed5-4330-97d4-73ce00b2d0c5}
   Set Set: Id {3062e440-988d-4ded-bb57-25ab087ce644}
   Property InTargetPosition: Id {13d374bf-abc5-4586-8edf-e398d810bb2b}
   Get Get: Id {f2945d22-f2f2-44ef-99b8-512ec77865b8}
   Set Set: Id {32bee957-6148-4a31-b07d-8d7ca43c83a4}
   Method Interlock: Id {72f66b07-eac8-4f48-a977-69dc5fa659a2}
   Method Logger: Id {7fb0d460-52d2-4ae2-accf-52e93bd858b3}
   Property McAxisState: Id {a5f0dcc8-191d-498e-b958-692049a1884c}
   Get Get: Id {419b3bc2-a2ce-4b0f-80d3-b1aaee4f3379}
   Set Set: Id {b3669996-ef61-4b88-a858-5b9a7358cb59}
   Method MotionParams: Id {d4d497ab-25de-4a2d-9f0c-7fd0abae8c76}
   Method MoveAbsolute: Id {67006bb1-1c73-49f6-ab52-7a06b1d0c294}
   Property MoveBusy: Id {d58c53d5-d71e-4dfb-81d9-c7fda2274825}
   Get Get: Id {0dc6e9a0-7a00-4339-8717-53ef63ce7bac}
   Set Set: Id {2b796103-4887-45ce-b787-f19ffce80544}
   Property MoveDone: Id {4dfc439a-a1c1-4c95-b749-95d177fa4901}
   Get Get: Id {8556348b-daa4-4c56-8993-087102c74a94}
   Set Set: Id {16c38ccc-bd1b-40f2-bbe5-f6aaca214440}
   Method MoveRelative: Id {274dd405-a068-4680-bb9e-fe5025f2f908}
   Method MoveVelocity: Id {ad5fd96d-9e69-45a4-b2a0-21317b75940d}
   Property PiezoErrorCode: Id {6909d919-bde9-446f-9642-d6b8f1850cfe}
   Get Get: Id {2ea8d926-6bc6-4780-b02a-0d0e439964a4}
   Set Set: Id {dec4dd39-3493-44de-bc51-b50700783e93}
   Method PostInterlocks: Id {0f2de4be-a2d5-40b5-bf2e-f13c48bf1447}
   Method Power: Id {634342db-4980-4103-96da-256cbacd69e1}
   Method ReadDriveErrors: Id {b0585027-4ae7-4117-8a3d-d9e1621fba78}
   Method ReadDriveParams: Id {91ee2260-ec1c-4238-9b91-9438ac703127}
   Method Reset: Id {ca77c887-2b90-4375-866f-a9f6ff5b335c}
   Method SetEnables: Id {8bb4d6f6-cdad-41b7-afa8-a970de274d07}
   Method SetServoOffParams: Id {a28d7e11-f485-4a60-bdef-9b0d673cfb42}
   Method StateMachine: Id {d963b9d7-d9e1-4a33-bb79-0f8a7e20b1de}
   Property Stopped: Id {d635cf6b-14dd-4bd9-916c-3698b86d0796}
   Get Get: Id {3dc0eca2-a01a-4678-8002-deb2233ad3a3}
   Set Set: Id {2a6dd676-a5db-4528-b3bd-d2f30f5c848e}
   Property stPzStage: Id {9f92815a-2a54-4642-bace-23982d7df851}
   Set Set: Id {c8f7e1d0-f544-4543-a5ce-d8889c56fbb7}
   Method SyncEpicsStatus: Id {0ec1ab11-3e34-4193-8590-6aaa07110b4c} *)
